TYPE ST_PneumaticAxisInputs :
STRUCT
    bEndSwitchValveOn AT %I*: BOOL; //End Switch valve on input
    bEndSwitchValveOff AT %I*: BOOL; //End Switch valve off input
    bValveOnManualOP1 AT %I*: BOOL; //Push button input to move to valve on position from Operator Panel 1
    bValveOffManualOP1 AT %I*: BOOL; //Push button input to move to valve off position from Operator Panel 1
    bValveOnManualOP2 AT %I*: BOOL; //Push button input to move to valve on position from Operator Panel 2
    bValveOffManualOP2 AT %I*: BOOL; //Push button input to move to valve off position from Operator Panel 2
END_STRUCT
END_TYPE

(* stored: Version 1.1.0.1
   DUT ST_PneumaticAxisInputs: Id {a13cd38f-3036-02f4-0651-ea4a97049122} *)
